% RSLogix 500 project PLC_INSTUCTIONS__1.RSS, saved by version 8.30.00.16 %
PROJECT "PLCFUNDA"    % processor: Bul.1763 MicroLogix 1100 Series B %

PROGRAM FILES
  LAD 2   26 rungs

DATA FILES
  O0 OUTPUT  4 elements
  I1 INPUT  6 elements
  S2 STATUS  66 elements
  B3 BINARY  1 elements
  T4 TIMER  3 elements
  C5 COUNTER  2 elements
  R6 CONTROL  1 elements
  N7 INTEGER  1 elements
  F8 FLOAT  1 elements

LADDER 2
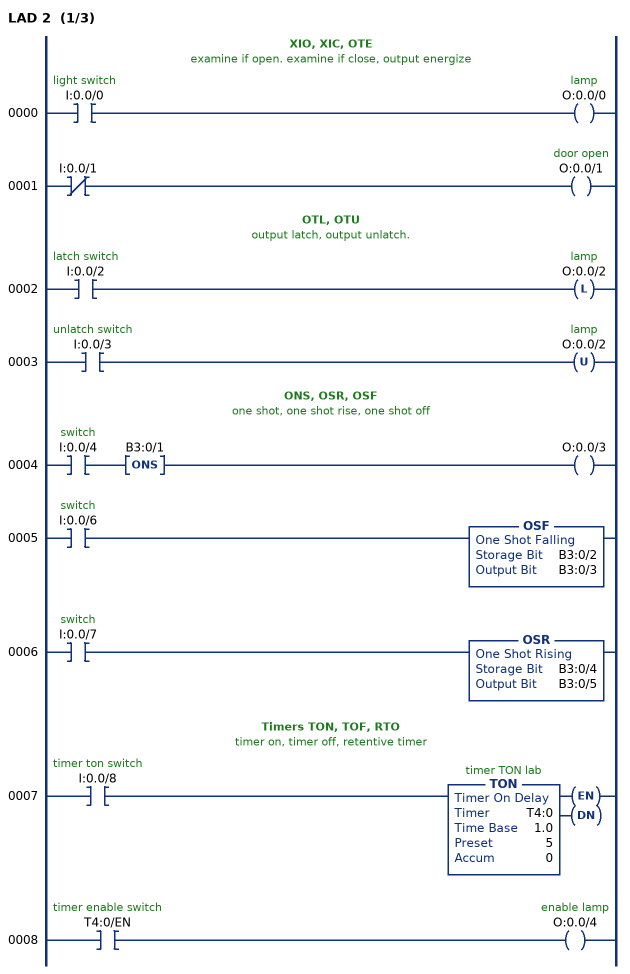
% Rung: 0 %
% TITLE: XIO, XIC, OTE %
% examine if open. examine if close, output energize %
SOR XIC I:0.0/0 OTE O:0.0/0 EOR
%   I:0.0/0  "light switch" %
%   O:0.0/0  "lamp" %
% Rung: 1 %
SOR XIO I:0.0/1 OTE O:0.0/1 EOR
%   O:0.0/1  "door open" %
% Rung: 2 %
% TITLE: OTL, OTU %
% output latch, output unlatch. %
SOR XIC I:0.0/2 OTL O:0.0/2 EOR
%   I:0.0/2  "latch switch" %
%   O:0.0/2  "lamp" %
% Rung: 3 %
SOR XIC I:0.0/3 OTU O:0.0/2 EOR
%   I:0.0/3  "unlatch switch" %
%   O:0.0/2  "lamp" %
% Rung: 4 %
% TITLE: ONS, OSR, OSF %
% one shot, one shot rise, one shot off %
SOR XIC I:0.0/4 ONS B3:0/1 OTE O:0.0/3 EOR
%   I:0.0/4  "switch" %
% Rung: 5 %
SOR XIC I:0.0/6 OSF B3:0/2 B3:0/3 EOR
%   I:0.0/6  "switch" %
% Rung: 6 %
SOR XIC I:0.0/7 OSR B3:0/4 B3:0/5 EOR
%   I:0.0/7  "switch" %
% Rung: 7 %
% TITLE: Timers TON, TOF, RTO %
% timer on, timer off, retentive timer %
SOR XIC I:0.0/8 TON T4:0 1.0 5 0 EOR
%   I:0.0/8  "timer ton switch" %
%   T4:0  "timer TON lab" %
% Rung: 8 %
SOR XIC T4:0/EN OTE O:0.0/4 EOR
%   T4:0/EN  "timer enable switch" %
%   O:0.0/4  "enable lamp" %

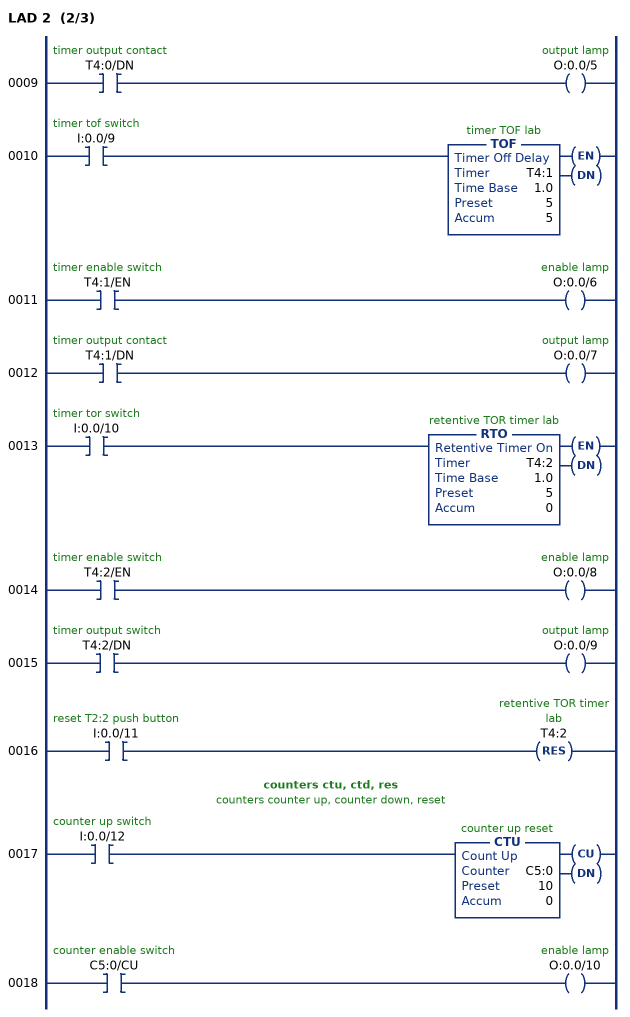
% Rung: 9 %
SOR XIC T4:0/DN OTE O:0.0/5 EOR
%   T4:0/DN  "timer output contact" %
%   O:0.0/5  "output lamp" %
% Rung: 10 %
SOR XIC I:0.0/9 TOF T4:1 1.0 5 5 EOR
%   I:0.0/9  "timer tof switch" %
%   T4:1  "timer TOF lab" %
% Rung: 11 %
SOR XIC T4:1/EN OTE O:0.0/6 EOR
%   T4:1/EN  "timer enable switch" %
%   O:0.0/6  "enable lamp" %
% Rung: 12 %
SOR XIC T4:1/DN OTE O:0.0/7 EOR
%   T4:1/DN  "timer output contact" %
%   O:0.0/7  "output lamp" %
% Rung: 13 %
SOR XIC I:0.0/10 RTO T4:2 1.0 5 0 EOR
%   I:0.0/10  "timer tor switch" %
%   T4:2  "retentive TOR timer lab" %
% Rung: 14 %
SOR XIC T4:2/EN OTE O:0.0/8 EOR
%   T4:2/EN  "timer enable switch" %
%   O:0.0/8  "enable lamp" %
% Rung: 15 %
SOR XIC T4:2/DN OTE O:0.0/9 EOR
%   T4:2/DN  "timer output switch" %
%   O:0.0/9  "output lamp" %
% Rung: 16 %
SOR XIC I:0.0/11 RES T4:2 EOR
%   I:0.0/11  "reset T2:2 push button" %
%   T4:2  "retentive TOR timer lab" %
% Rung: 17 %
% TITLE: counters ctu, ctd, res %
% counters counter up, counter down, reset %
SOR XIC I:0.0/12 CTU C5:0 10 0 EOR
%   I:0.0/12  "counter up switch" %
%   C5:0  "counter up reset" %
% Rung: 18 %
SOR XIC C5:0/CU OTE O:0.0/10 EOR
%   C5:0/CU  "counter enable switch" %
%   O:0.0/10  "enable lamp" %

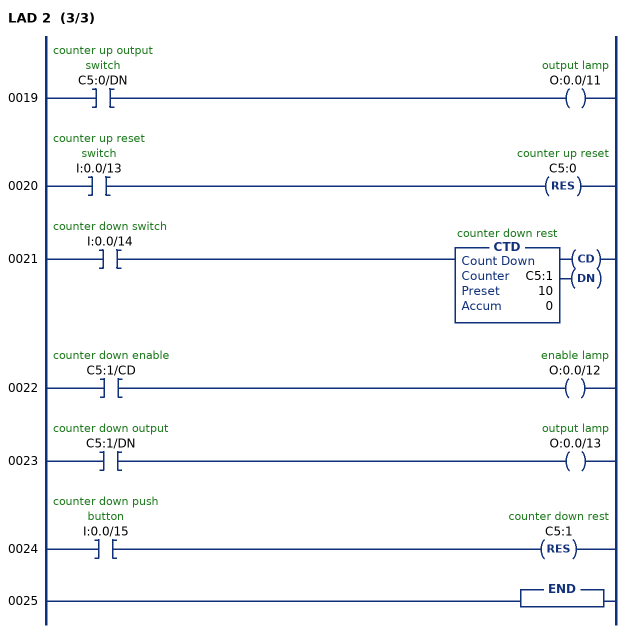
% Rung: 19 %
SOR XIC C5:0/DN OTE O:0.0/11 EOR
%   C5:0/DN  "counter up output switch" %
%   O:0.0/11  "output lamp" %
% Rung: 20 %
SOR XIC I:0.0/13 RES C5:0 EOR
%   I:0.0/13  "counter up reset switch" %
%   C5:0  "counter up reset" %
% Rung: 21 %
SOR XIC I:0.0/14 CTD C5:1 10 0 EOR
%   I:0.0/14  "counter down switch" %
%   C5:1  "counter down rest" %
% Rung: 22 %
SOR XIC C5:1/CD OTE O:0.0/12 EOR
%   C5:1/CD  "counter down enable" %
%   O:0.0/12  "enable lamp" %
% Rung: 23 %
SOR XIC C5:1/DN OTE O:0.0/13 EOR
%   C5:1/DN  "counter down output" %
%   O:0.0/13  "output lamp" %
% Rung: 24 %
SOR XIC I:0.0/15 RES C5:1 EOR
%   I:0.0/15  "counter down push button" %
%   C5:1  "counter down rest" %
% Rung: 25 %
SOR END EOR

OTHER DOCUMENTED ADDRESSES
  O:0  "one shot"

DATA TABLE (non-zero values as saved)
DATA T4
% .PRE .ACC %
% T4:0 % 5 0
% T4:1 % 5 5
% T4:2 % 5 0
DATA C5
% .PRE .ACC %
% C5:0 % 10 0
% C5:1 % 10 0
